INTERFACE I_BA_MyWeatherStation EXTENDS I_BA_Publisher

PROPERTY Brightness : REAL
GET
END_GET
END_PROPERTY

PROPERTY Error : BOOL
GET
END_GET
END_PROPERTY

PROPERTY Humidity : REAL
GET
END_GET
END_PROPERTY

PROPERTY Latitude : REAL
GET
END_GET
END_PROPERTY

PROPERTY Longitude : REAL
GET
END_GET
END_PROPERTY

PROPERTY Ready : BOOL
GET
END_GET
END_PROPERTY

PROPERTY WeatherTemperature : REAL
GET
END_GET
END_PROPERTY

PROPERTY WindDirection : REAL
GET
END_GET
END_PROPERTY

PROPERTY WindSpeed : REAL
GET
END_GET
END_PROPERTY

END_INTERFACE

(* stored: Version 1.1.0.1, ProductVersion 3.1.4024.5
   Itf I_BA_MyWeatherStation: Id {a541aedf-0be9-4218-938d-5a0290287e6a}
   Folder Management: Id {350159f5-30c7-43b7-a1bd-601c4ecc03b2}
   Folder Properties: Id {043a9c97-b628-467d-9e4d-9a0dd644f770}
   Folder Properties: Id {094b92cb-adeb-474a-a6be-99cdf2ee662f}
   Property Brightness: Id {6e669859-e69e-4060-a1a1-f061fcc8a293}
   Get Get: Id {ed87f8a8-200e-4833-80ce-d1794157e62e}
   Property Error: Id {e2b2bba7-c317-43ee-8495-01bd99af4304}
   Get Get: Id {1f900cec-e275-4327-b8c2-7f6f1ed374b2}
   Property Humidity: Id {caf869a8-0ab0-4e37-b928-a5ef97404098}
   Get Get: Id {31bc0818-5e49-406d-bfc8-068ee7eed363}
   Property Latitude: Id {187741d3-c152-4e3a-be13-06ce48f4efea}
   Get Get: Id {f9bf9f9a-3576-40da-8bde-11144ddde644}
   Property Longitude: Id {63433b94-c631-4610-b415-3cdf751dcf34}
   Get Get: Id {becae2b9-2360-458e-ba6f-30762e3a61e9}
   Property Ready: Id {30c39fdb-9ef5-446f-b328-18e3e4122697}
   Get Get: Id {657e7cd7-7524-4c0e-b92d-0e70220bcdc1}
   Property WeatherTemperature: Id {ca439baa-683c-465a-a50d-80be3262a9e7}
   Get Get: Id {cf28c190-fb6b-4715-bc22-8157e04bc0b5}
   Property WindDirection: Id {978d28e3-3d6b-4813-93b1-ce74be2b3681}
   Get Get: Id {fb01582c-cbd2-407d-9e4f-31f46ebcca09}
   Property WindSpeed: Id {a0f2a058-e714-4d0a-9501-aac13cdc34d8}
   Get Get: Id {fc9d5796-233b-483b-9680-43f8d56f640d} *)
